# EPICS autosave request: mrfApp/Db/evr-delay-compensation.inc.req
$(P)$(R)DelayComp:Enabled.VAL
$(P)$(R)DelayComp:TargetDelay.VAL
